# EPICS substitutions: snmp2/iocBoot/iocsnmp2/brocade.substitutions
file "${RAON_SITEAPPS}/snmp2/db/brocade.db"
{
pattern
{SYS, SUBSYS, DEV, N, P, V2C, HOST, COM, T}
{CTRL, NET, SW, 005, 1, SNMP_VERSION_2c, 192.168.1.20, public, 1}
{CTRL, NET, SW, 005, 2, SNMP_VERSION_2c, 192.168.1.20, public, 2}
{CTRL, NET, SW, 005, 3, SNMP_VERSION_2c, 192.168.1.20, public, 3}
{CTRL, NET, SW, 005, 4, SNMP_VERSION_2c, 192.168.1.20, public, 4}
{CTRL, NET, SW, 005, 5, SNMP_VERSION_2c, 192.168.1.20, public, 5}
{CTRL, NET, SW, 005, 6, SNMP_VERSION_2c, 192.168.1.20, public, 6}
{CTRL, NET, SW, 005, 7, SNMP_VERSION_2c, 192.168.1.20, public, 7}
{CTRL, NET, SW, 005, 8, SNMP_VERSION_2c, 192.168.1.20, public, 8}
{CTRL, NET, SW, 005, 9, SNMP_VERSION_2c, 192.168.1.20, public, 9}
{CTRL, NET, SW, 005, 10, SNMP_VERSION_2c, 192.168.1.20, public, 10}
{CTRL, NET, SW, 005, 11, SNMP_VERSION_2c, 192.168.1.20, public, 11}
{CTRL, NET, SW, 005, 12, SNMP_VERSION_2c, 192.168.1.20, public, 12}
{CTRL, NET, SW, 005, 13, SNMP_VERSION_2c, 192.168.1.20, public, 13}
{CTRL, NET, SW, 005, 14, SNMP_VERSION_2c, 192.168.1.20, public, 14}
{CTRL, NET, SW, 005, 15, SNMP_VERSION_2c, 192.168.1.20, public, 15}
{CTRL, NET, SW, 005, 16, SNMP_VERSION_2c, 192.168.1.20, public, 16}
{CTRL, NET, SW, 005, 17, SNMP_VERSION_2c, 192.168.1.20, public, 17}
{CTRL, NET, SW, 005, 18, SNMP_VERSION_2c, 192.168.1.20, public, 18}
{CTRL, NET, SW, 005, 19, SNMP_VERSION_2c, 192.168.1.20, public, 19}
{CTRL, NET, SW, 005, 20, SNMP_VERSION_2c, 192.168.1.20, public, 20}
{CTRL, NET, SW, 005, 21, SNMP_VERSION_2c, 192.168.1.20, public, 21}
{CTRL, NET, SW, 005, 22, SNMP_VERSION_2c, 192.168.1.20, public, 22}
{CTRL, NET, SW, 005, 23, SNMP_VERSION_2c, 192.168.1.20, public, 23}
{CTRL, NET, SW, 005, 24, SNMP_VERSION_2c, 192.168.1.20, public, 24}
{CTRL, NET, SW, 005, 25, SNMP_VERSION_2c, 192.168.1.20, public, 25}
{CTRL, NET, SW, 005, 26, SNMP_VERSION_2c, 192.168.1.20, public, 26}
{CTRL, NET, SW, 005, 27, SNMP_VERSION_2c, 192.168.1.20, public, 27}
{CTRL, NET, SW, 005, 28, SNMP_VERSION_2c, 192.168.1.20, public, 28}
{CTRL, NET, SW, 005, 29, SNMP_VERSION_2c, 192.168.1.20, public, 29}
{CTRL, NET, SW, 005, 30, SNMP_VERSION_2c, 192.168.1.20, public, 30}
{CTRL, NET, SW, 005, 31, SNMP_VERSION_2c, 192.168.1.20, public, 31}
{CTRL, NET, SW, 005, 32, SNMP_VERSION_2c, 192.168.1.20, public, 32}
{CTRL, NET, SW, 005, 33, SNMP_VERSION_2c, 192.168.1.20, public, 33}
{CTRL, NET, SW, 005, 34, SNMP_VERSION_2c, 192.168.1.20, public, 34}
{CTRL, NET, SW, 005, 35, SNMP_VERSION_2c, 192.168.1.20, public, 35}
{CTRL, NET, SW, 005, 36, SNMP_VERSION_2c, 192.168.1.20, public, 36}
{CTRL, NET, SW, 005, 37, SNMP_VERSION_2c, 192.168.1.20, public, 37}
{CTRL, NET, SW, 005, 38, SNMP_VERSION_2c, 192.168.1.20, public, 38}
{CTRL, NET, SW, 005, 39, SNMP_VERSION_2c, 192.168.1.20, public, 39}
{CTRL, NET, SW, 005, 40, SNMP_VERSION_2c, 192.168.1.20, public, 40}
{CTRL, NET, SW, 005, 41, SNMP_VERSION_2c, 192.168.1.20, public, 41}
{CTRL, NET, SW, 005, 42, SNMP_VERSION_2c, 192.168.1.20, public, 42}
{CTRL, NET, SW, 005, 43, SNMP_VERSION_2c, 192.168.1.20, public, 43}
{CTRL, NET, SW, 005, 44, SNMP_VERSION_2c, 192.168.1.20, public, 44}
{CTRL, NET, SW, 005, 45, SNMP_VERSION_2c, 192.168.1.20, public, 45}
{CTRL, NET, SW, 005, 46, SNMP_VERSION_2c, 192.168.1.20, public, 46}
{CTRL, NET, SW, 005, 47, SNMP_VERSION_2c, 192.168.1.20, public, 47}
{CTRL, NET, SW, 005, 48, SNMP_VERSION_2c, 192.168.1.20, public, 48}
